INTERFACE I_MotionAxisStage

END_INTERFACE

(* stored: Version 1.1.0.1
   Itf I_MotionAxisStage: Id {dfb7fe95-39d5-4c28-92ce-bc7af482abb6} *)
